Staubli VAL3: create.pgx

public program create(num x_nConvNum)
  local num l_nError
  local num l_nValue
begin
  call init(x_nConvNum,l_nError)
  if l_nError==0
    //
    call enc:getResolution(l_nValue)
    if roundDown(l_nValue)!=roundDown(nENCRESOLUTION)
      call enc:setResolution(nENCRESOLUTION)
      popUpMsg("Warning: a change has been detected in the encoder resolution.  The calibration of your conveyor may be not valid anymore")
    else
    endIf
    // Start encoder
    call enc:create(x_nConvNum,sTASK[1])
    // Start management of conveyor queue
    taskCreate sTASK[0]+toString("",x_nConvNum),100,conveyor()
    //Start Detection
    call det:create(x_nConvNum,sTASK[2])
  endIf
end
